// Block: A0301_Spintore_Lat_PERS

DATA_BLOCK A0301_Spintore_Lat_PERS
VERSION : 0.1
   NON_RETAIN
   VAR
      Spin_Lat_1 : Struct
         Par : Analogic_SensorManagement_Par;
         Data : Struct
            Sens : Analogic_SensorManagement_Data;
            HMI : HMI_Preset;
         END_STRUCT;
         Par_Mach : A0301_Mach_Sens_Par;
      END_STRUCT;
      Spin_Lat_2 : Struct
         Par : Analogic_SensorManagement_Par;
         Data : Struct
            Sens : Analogic_SensorManagement_Data;
            HMI : HMI_Preset;
         END_STRUCT;
         Par_Mach : A0301_Mach_Sens_Par;
      END_STRUCT;
   END_VAR

BEGIN
   // No initialization required
END_DATA_BLOCK
